FUNCTION_BLOCK integEC (* Ground-truth reference: generic time-based integrator (physical cylinder position model) *)
  (* Standard: 61499-2; Description: Educational reference, ported for the Meisterschulen am Ostbahnhof IEC 61499 training repository. Original design (c) nxtControl GmbH, from the UniversalAutomation.org 'IEC 61499: primer course' curriculum exercise Final.sln (also present in the LiftingLuggage_*.sln/Starter.sln exercises), IEC61499/integEC.fbt - included here under the same educational-use terms as the rest of that curriculum. This port: Copyright (c) 2026 Meisterschulen am Ostbahnhof, EPL-2.0, https://www.eclipse.org/legal/epl-2.0/ *)
  (* Version 0.0, 2007-06-14, milos, nxtControl GmbH, Original EAE/nxtControl design (Template), source: Final.sln (identical copies in LiftingLuggage_*.sln, Starter.sln) *)
  (* Version 1.0, 2026-09-03, Franz Höpfinger, Meisterschulen am Ostbahnhof, Ported from EAE/nxtControl format (LibraryElement.dtd, ST as an attribute with escapes) to 4diac's FBType XSD (ST as CDATA). Interface, ECC, and both algorithms otherwise unchanged. Part of the CylinderH continuous-simulation reference - see ContinuousCylinderSimulation.md *)
  (* Version 1.1, 2026-09-03, Franz Höpfinger, Meisterschulen am Ostbahnhof, PR #160 review feedback: INIT/INITO must be Type=EInit (were Type=Event) - fixed, With-Var lists unchanged *)
  (* Version 1.2, 2026-09-03, Franz Höpfinger, Meisterschulen am Ostbahnhof, PR #160 review feedback (coderabbitai): documented that TRIP/P_TRIP are practically unreachable due to ECC transition declaration order (execIntegration's C_CYCLE[NOT error] always wins first), inherited unchanged from the original nxtControl source. Not fixed - no effect on CylinderHCore.fbt, which never wires these outputs; would need a real ECC restructuring *)
  PACKAGE Meins::DesingPatterns::ContinuousCylinderSimulation;
  (* Documentation:
  Ground-truth reference, not a Vyatkin Module 6 slide pattern. Generic time-based integrator, ported as-is from the UniversalAutomation.org "IEC 61499: primer course" curriculum (Final.sln, IEC61499/integEC.fbt, original format: EAE/nxtControl LibraryElement.dtd). Used by CylinderHCore.fbt in this folder as the physical cylinder's position model: on every C_CYCLE tick it integrates pv1/pv2 (the two extend/retract drive signals) over cycleTime, optionally clamped to [minValue, maxValue], producing total (raw position) and out (position, or distance-to-setpoint if integType=1).
   Renamed state vs. the original: the original names its reset state RESET, identical to its own RESET event. Renamed to RESET_ST here purely as a precaution against a same-name event/state clash (not confirmed to actually be a problem in 4diac, just untested either way) - no functional change.
   Known limitation, inherited from the original (PR #160 review, coderabbitai): TRIP/P_TRIP are practically unreachable. IEC 61499 ECC evaluates a state's outgoing transitions in declaration order and takes the first whose condition is true; START -> execIntegration (C_CYCLE[NOT error]) is declared before START -> raiseTrip/ raisePTrip, and its condition is true on every C_CYCLE as long as error=FALSE - so the threshold transitions never get evaluated during normal operation. This exact transition order already exists unchanged in the original nxtControl source. Not fixed here: it is a real ECC restructuring (a dedicated calculation state, then mutually exclusive threshold checks afterward), and it has no effect on CylinderHCore.fbt in this folder, which never wires Model.TRIP/ Model.P_TRIP to anything. Worth fixing if this block is ever reused somewhere that actually needs the trip outputs.
  *)
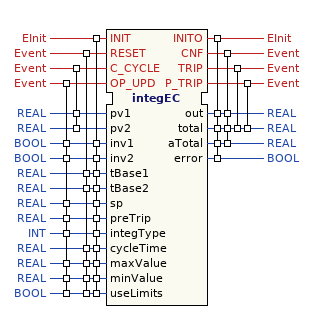
  EVENT_INPUT
    INIT : EInit WITH inv1, inv2, tBase1, tBase2, sp, preTrip, integType, cycleTime, maxValue, minValue, useLimits; (* Initialization Request *)
    RESET WITH tBase1, tBase2, cycleTime, maxValue, minValue, useLimits; (* reset integrator *)
    C_CYCLE WITH pv1, pv2; (* cycle calculation call *)
    OP_UPD WITH sp, preTrip, inv1, inv2, integType, maxValue, minValue, useLimits; (* new operator parameter *)
  END_EVENT
  EVENT_OUTPUT
    INITO : EInit WITH out, total, aTotal, error; (* Initialization Confirm *)
    CNF WITH out, total, aTotal; (* Execution Confirmation *)
    TRIP WITH total; (* total >= sp *)
    P_TRIP WITH total; (* preTrip > (sp - total) *)
  END_EVENT
  VAR_INPUT
    pv1 : REAL := 0.0; (* pv1 to integrate *)
    pv2 : REAL := 0.0; (* pv2 to integrate *)
    inv1 : BOOL := FALSE; (* invert (multiply with -1) pv1 *)
    inv2 : BOOL := FALSE; (* invert (multiply with -1) pv2 *)
    tBase1 : REAL := 3600.0; (* timebase of pv1 [s] *)
    tBase2 : REAL := 3600.0; (* timebase of pv2 [s] *)
    sp : REAL := 0.0; (* setpoint of integrator *)
    preTrip : REAL := 0.0; (* distance to setpoint for preTrip to set *)
    integType : INT := 0; (* integration Type *)
    cycleTime : REAL := 1.0; (* cycle Time for calculation *)
    maxValue : REAL;
    minValue : REAL;
    useLimits : BOOL;
  END_VAR
  VAR_OUTPUT
    out : REAL := 0.0; (* out value (depends on integType) *)
    total : REAL := 0.0; (* integrated summation of all pv *)
    aTotal : REAL := 0.0; (* signed integrated summation of pv1/tBase1+pv2/tBase2, without inv1/inv2 correction (despite the name, calcTotal never applies ABS() - an inconsistency already present in the original nxtControl source, preserved as-is here) *)
    error : BOOL := FALSE; (* error detected *)
  END_VAR
  VAR
    sumPv : REAL := 0.0; (* time based sum of pv (with inv correction) *)
  END_VAR
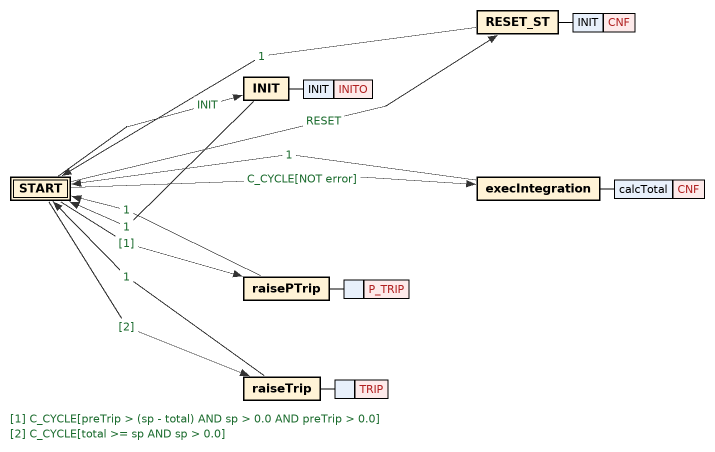
  EC_STATES
    START; (* Initial State *)
    INIT : INIT -> INITO; (* Initialization *)
    execIntegration : calcTotal -> CNF; (* Normal execution: one integration step *)
    raiseTrip : -> TRIP; (* total reached the setpoint - KNOWN LIMITATION: unreachable while error=FALSE, see Documentation *)
    raisePTrip : -> P_TRIP; (* total is within preTrip of the setpoint - KNOWN LIMITATION: unreachable while error=FALSE, see Documentation *)
    RESET_ST : INIT -> CNF; (* Reset the integrator *)
  END_STATES
  EC_TRANSITIONS
    START TO INIT := INIT;
    INIT TO START := 1;
    START TO execIntegration := C_CYCLE[NOT error];
    execIntegration TO START := 1;
    START TO raiseTrip := C_CYCLE[total >= sp AND sp > 0.0];
    raiseTrip TO START := 1;
    START TO raisePTrip := C_CYCLE[preTrip > (sp - total) AND sp > 0.0 AND preTrip > 0.0];
    raisePTrip TO START := 1;
    START TO RESET_ST := RESET;
    RESET_ST TO START := 1;
  END_TRANSITIONS
  ALGORITHM INIT IN ST: (* Reset the integrator outputs *)
out := 0.0;
total := 0.0;
aTotal := 0.0;
error := (tBase1 <= 0.0) OR (tBase2 <= 0.0) OR (cycleTime <= 0.0);
  END_ALGORITHM
  ALGORITHM calcTotal IN ST: (* One integration step over cycleTime *)
aTotal := aTotal + cycleTime * (pv1/tBase1 + pv2/tBase2);

IF inv1 THEN
	sumPv := pv1/tBase1 * -1.0;
ELSE
	sumPv := pv1/tBase1;
END_IF;
IF inv2 THEN
	sumPv := sumPv + pv2/tBase2 * -1.0;
ELSE
	sumPv := sumPv + pv2/tBase2;
END_IF;

total := total + cycleTime * sumPv;

IF useLimits THEN
	total := LIMIT(minValue, total, maxValue);
END_IF;

IF integType = 1 AND sp > 0.0 THEN
	out := sp-total;
ELSE
	out := total;
END_IF;
  END_ALGORITHM
END_FUNCTION_BLOCK
